// TIA Portal V17 export
// export: Created 2025-03-07T09:19:45.6758069Z, ExportSetting WithDefaults, DisplayName Totally Integrated Automation Portal, DisplayVersion V17 Update 8, DisplayName TIA Portal Openness, DisplayVersion V17 Update 8, DisplayName TIA Portal Version Control Interface, DisplayVersion V17, DisplayName SINAMICS Startdrive Advanced, DisplayVersion V17 SP2, DisplayName SINAMICS Startdrive G110M, G120, G120C, G120D, G120P, G115D, DisplayVersion V17 SP2, DisplayName SINAMICS Startdrive G130, G150, S120, S150, SINAMICS MV, S210, DisplayVersion V17 SP2, DisplayName STEP 7 Professional, DisplayVersion V17 Update 8, DisplayName SINUMERIK ONE STEP 7 Toolbox, DisplayVersion V17 Update 12, DisplayName SINUMERIK 840D sl STEP 7 Toolbox, DisplayVersion V17 Update 12, DisplayName STEP 7 Safety, DisplayVersion V17 Update 6, DisplayName WinCC Advanced, DisplayVersion V17 Update 8
TYPE "SEQUENCE"
// stored: IsFailsafeCompliant false
   STRUCT
      GENERAL_CONDITIONS : Bool;   // UNIT 01L CYCLE SEQUENCE GENERAL CONDITIONS / GENERAL CONDITIONS
      INITIAL_CONDITIONS : Bool;   // UNIT 01L CYCLE SEQUENCE INITIAL CONDITIONS / INITIAL CONDITIONS
      REQUEST : Bool;   // UNIT 01L START CYCLE SEQUENCE REQUEST / REQUEST
      REQUEST_PULSE : Bool;   // UNIT 01L CYCLE SEQUENCE REQUEST PULSE / REQUEST PULSE
      COMMAND : Bool;   // UNIT 01L CYCLE SEQUENCE COMMAND / COMMAND
      COMMAND_PULSE : Bool;   // UNIT 01L CYCLE SEQUENCE COMMAND PULSE / COMMAND PULSE
      RUNNING : Bool;   // UNIT 01L CYCLE SEQUENCE IN PROCESS / RUNNING
      SPARE : Bool;   // SPARE
      STEP_1 : Bool;   // UNIT 01L CYCLE SEQUENCE STEP 1 / STEP 1
      STEP_2 : Bool;   // UNIT 01L CYCLE SEQUENCE STEP 2 / STEP 2
      STEP_3 : Bool;   // UNIT 01L CYCLE SEQUENCE STEP 3 / STEP 3
      STEP_4 : Bool;   // UNIT 01L CYCLE SEQUENCE STEP 4 / STEP 4
      STEP_5 : Bool;   // UNIT 01L CYCLE SEQUENCE STEP 5 / STEP 5
      STEP_6 : Bool;   // UNIT 01L CYCLE SEQUENCE STEP 6 / STEP 6
      STEP_7 : Bool;   // UNIT 01L CYCLE SEQUENCE STEP 7 / STEP 7
      STEP_8 : Bool;   // UNIT 01L CYCLE SEQUENCE STEP 8 / STEP 8
      STEP_9 : Bool;   // UNIT 01L CYCLE SEQUENCE STEP 9 / STEP 9
      STEP_10 : Bool;   // UNIT 01L CYCLE SEQUENCE STEP 10 / STEP 10
      STEP_11 : Bool;   // UNIT 01L CYCLE SEQUENCE STEP 11 / STEP 11
      STEP_12 : Bool;   // UNIT 01L CYCLE SEQUENCE STEP 12 / STEP 12
      STEP_13 : Bool;   // UNIT 01L CYCLE SEQUENCE STEP 13 / STEP 13
      STEP_14 : Bool;   // UNIT 01L CYCLE SEQUENCE STEP 14 / STEP 14
      STEP_15 : Bool;   // UNIT 01L CYCLE SEQUENCE STEP 15 / STEP 15
      STEP_16 : Bool;   // UNIT 01L CYCLE SEQUENCE STEP 16 / STEP 16
      STEP_17 : Bool;   // STEP 17
      STEP_18 : Bool;   // STEP 18
      STEP_19 : Bool;   // STEP 19
      STEP_20 : Bool;   // STEP 20
      STEP_21 : Bool;   // STEP 21
      STEP_22 : Bool;   // STEP 22
      STEP_23 : Bool;   // STEP 23
      STEP_24 : Bool;   // STEP 24
      STEP_25 : Bool;   // STEP 25
      STEP_26 : Bool;   // STEP 26
      STEP_27 : Bool;   // STEP 27
      STEP_28 : Bool;   // STEP 28
      STEP_29 : Bool;   // STEP 29
      STEP_30 : Bool;   // STEP 30
      STEP_31 : Bool;   // STEP 31
      STEP_32 : Bool;   // STEP 32
      RESET_PLC_AND_CNC : Bool;   // UNIT 01L CYCLE SEQUENCE RESET PLC AND CNC / RESET PLC AND CNC
      HMI_SEMI_REQUEST : Bool;   // HMI PUSHBUTTON SEMI REQUEST
      SEMI_AUTO_REQUEST : Bool;   // UNIT 01L CYCLE SEQUENCE SEMI AUTO REQUEST / SEMI AUTO REQUEST
      SEMI_AUTO_REQUEST_PULSE : Bool;   // UNIT 01L CYCLE SEQUENCE SEMI AUTO REQUEST / SEMI AUTO REQUEST PULSE
      AUTO_REQUEST : Bool;   // UNIT 01L CYCLE SEQUENCE AUTO REQUEST / AUTO REQUEST
      DONE : Bool;   // UNIT 01L CYCLE SEQUENCE DONE / DONE
      TIME_EXCEEDED : Bool;   // UNIT 01L CYCLE SEQUENCE TIME EXCEEDED / TIME EXCEEDED ALARM
      PREALARM : Bool;   // UNIT 01L CYCLE SEQUENCE PREALARM / PREALARM
      AUX0 : Bool;   // UNIT 01L CYCLE SEQUENCE AUX0 / AUXILIARY 0
      AUX1 : Bool;   // UNIT 01L CYCLE SEQUENCE AUX1 / AUXILIARY 1
      AUX2 : Bool;   // UNIT 01L CYCLE SEQUENCE AUX2 / AUXILIARY 2
      AUX3 : Bool;   // UNIT 01L CYCLE SEQUENCE AUX3 / AUXILIARY 3
      AUX5 : Bool;   // UNIT 01L CYCLE SEQUENCE AUX5 / AUXILIARY 5
      AUX6 : Bool;   // UNIT 01L CYCLE SEQUENCE AUX6 / AUXILIARY 6
      AUX7 : Bool;   // UNIT 01L CYCLE SEQUENCE AUX7 / AUXILIARY 7
      PREALARM_GONE : Bool;   // UNIT 01L CYCLE SEQUENCE PREALARM GONE / PREALARM GONE
      GENERAL_CONDITIONS_HELP : Bool;   // UNIT 01L CYCLE SEQUENCE GENERAL CONDITIONS HELP / GENERAL CONDITIONS HELP
      INITIAL_CONDITIONS_HELP : Bool;   // UNIT 01L CYCLE SEQUENCE INITIAL CONDITIONS HELP / INITIAL CONDITIONS HELP
      TIMER_TIME_EXCEED { S7_SetPoint := 'True'} : TON_TIME;   // TIME EXCEEDED TIMER
   END_STRUCT;
END_TYPE
